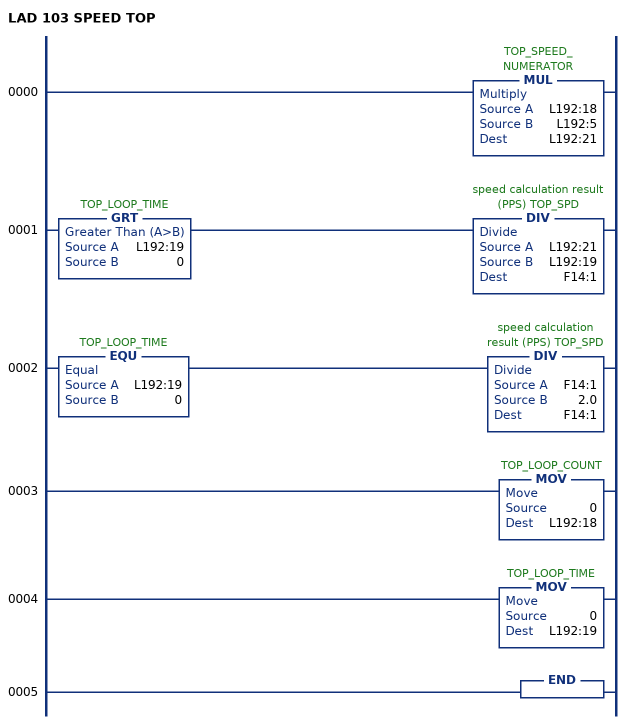
% Rung: 0 %
SOR MUL L192:18 L192:5 L192:21 EOR
%   L192:18  TOP_LOOP_COUNT %
%   L192:5  TKS_PER_SECOND %
%   L192:21  TOP_SPEED_NUMERATOR %
% Rung: 1 %
SOR GRT L192:19 0 DIV L192:21 L192:19 F14:1 EOR
%   L192:19  TOP_LOOP_TIME %
%   L192:21  TOP_SPEED_NUMERATOR %
%   F14:1  TOP_SPD  "speed calculation result (PPS)" %
% Rung: 2 %
SOR EQU L192:19 0 DIV F14:1 2.0 F14:1 EOR
%   L192:19  TOP_LOOP_TIME %
%   F14:1  TOP_SPD  "speed calculation result (PPS)" %
% Rung: 3 %
SOR MOV 0 L192:18 EOR
%   L192:18  TOP_LOOP_COUNT %
% Rung: 4 %
SOR MOV 0 L192:19 EOR
%   L192:19  TOP_LOOP_TIME %
% Rung: 5 %
SOR END EOR

LADDER 104 "P BOT"    % high speed %
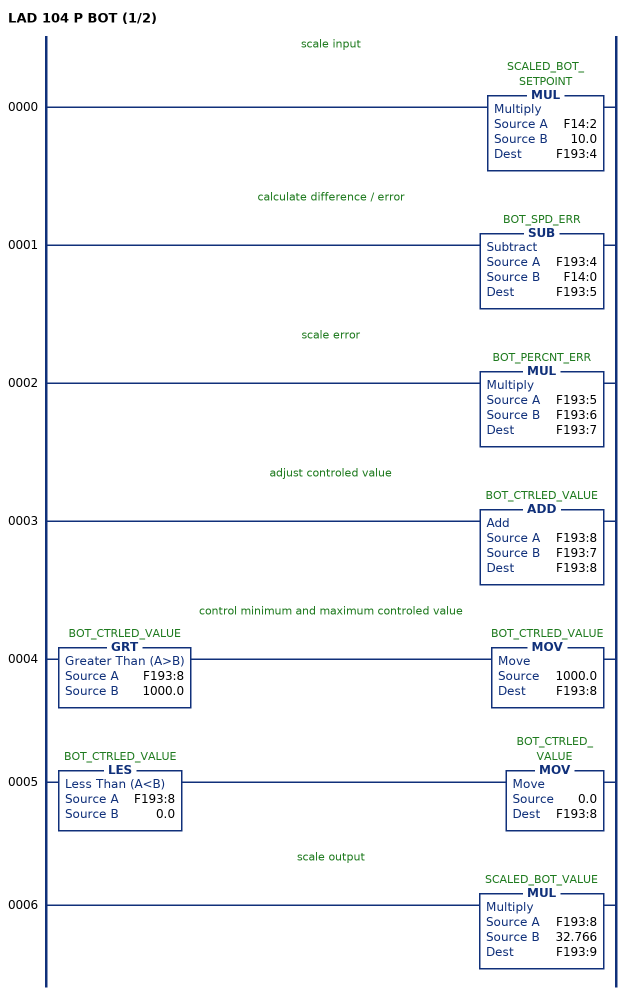
% Rung: 0 %
% scale input %
SOR MUL F14:2 10.0 F193:4 EOR
%   F14:2  BOT_SPD_SETPOINT %
%   F193:4  SCALED_BOT_SETPOINT %
% Rung: 1 %
% calculate difference / error %
SOR SUB F193:4 F14:0 F193:5 EOR
%   F193:4  SCALED_BOT_SETPOINT %
%   F14:0  BOT_SPD  "speed calculation result (PPS)" %
%   F193:5  BOT_SPD_ERR %
% Rung: 2 %
% scale error %
SOR MUL F193:5 F193:6 F193:7 EOR
%   F193:5  BOT_SPD_ERR %
%   F193:6  BOT_FDBK_RATIO %
%   F193:7  BOT_PERCNT_ERR %
% Rung: 3 %
% adjust controled value %
SOR ADD F193:8 F193:7 F193:8 EOR
%   F193:8  BOT_CTRLED_VALUE %
%   F193:7  BOT_PERCNT_ERR %
% Rung: 4 %
% control minimum and maximum controled value %
SOR GRT F193:8 1000.0 MOV 1000.0 F193:8 EOR
%   F193:8  BOT_CTRLED_VALUE %
% Rung: 5 %
SOR LES F193:8 0.0 MOV 0.0 F193:8 EOR
%   F193:8  BOT_CTRLED_VALUE %
% Rung: 6 %
% scale output %
SOR MUL F193:8 32.766 F193:9 EOR
%   F193:8  BOT_CTRLED_VALUE %
%   F193:9  SCALED_BOT_VALUE %

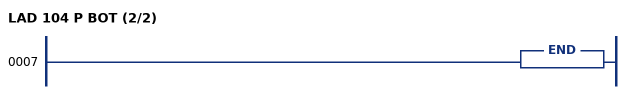
% Rung: 7 %
SOR END EOR

LADDER 105 "P TOP"    % high speed %
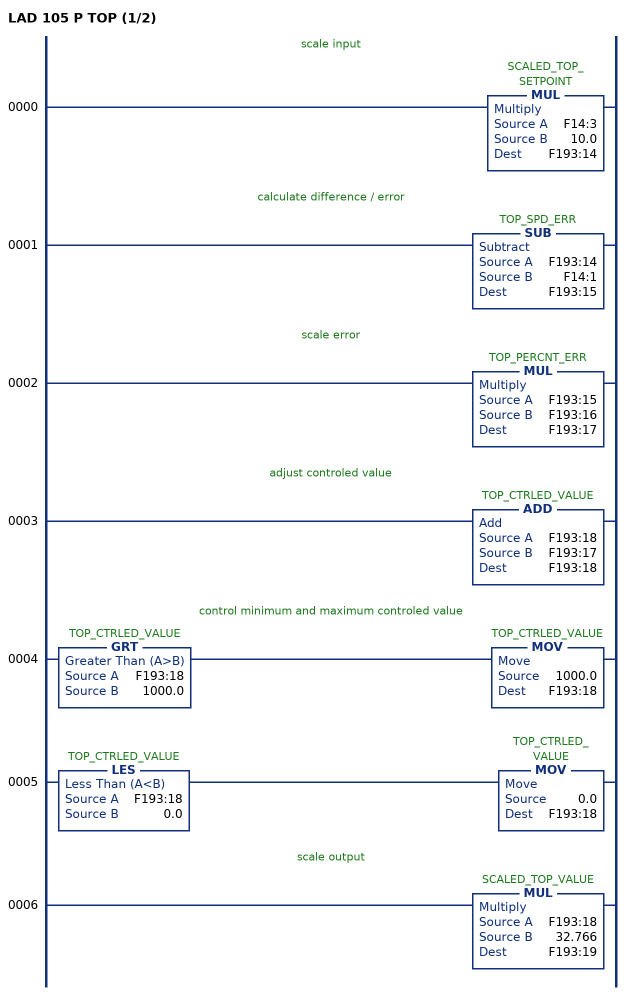
% Rung: 0 %
% scale input %
SOR MUL F14:3 10.0 F193:14 EOR
%   F14:3  TOP_SPD_SETPOINT %
%   F193:14  SCALED_TOP_SETPOINT %
% Rung: 1 %
% calculate difference / error %
SOR SUB F193:14 F14:1 F193:15 EOR
%   F193:14  SCALED_TOP_SETPOINT %
%   F14:1  TOP_SPD  "speed calculation result (PPS)" %
%   F193:15  TOP_SPD_ERR %
% Rung: 2 %
% scale error %
SOR MUL F193:15 F193:16 F193:17 EOR
%   F193:15  TOP_SPD_ERR %
%   F193:16  TOP_FDBK_RATIO %
%   F193:17  TOP_PERCNT_ERR %
% Rung: 3 %
% adjust controled value %
SOR ADD F193:18 F193:17 F193:18 EOR
%   F193:18  TOP_CTRLED_VALUE %
%   F193:17  TOP_PERCNT_ERR %
% Rung: 4 %
% control minimum and maximum controled value %
SOR GRT F193:18 1000.0 MOV 1000.0 F193:18 EOR
%   F193:18  TOP_CTRLED_VALUE %
% Rung: 5 %
SOR LES F193:18 0.0 MOV 0.0 F193:18 EOR
%   F193:18  TOP_CTRLED_VALUE %
% Rung: 6 %
% scale output %
SOR MUL F193:18 32.766 F193:19 EOR
%   F193:18  TOP_CTRLED_VALUE %
%   F193:19  SCALED_TOP_VALUE %

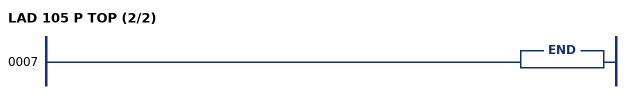
% Rung: 7 %
SOR END EOR

LADDER 110 "SHIFT BOT"
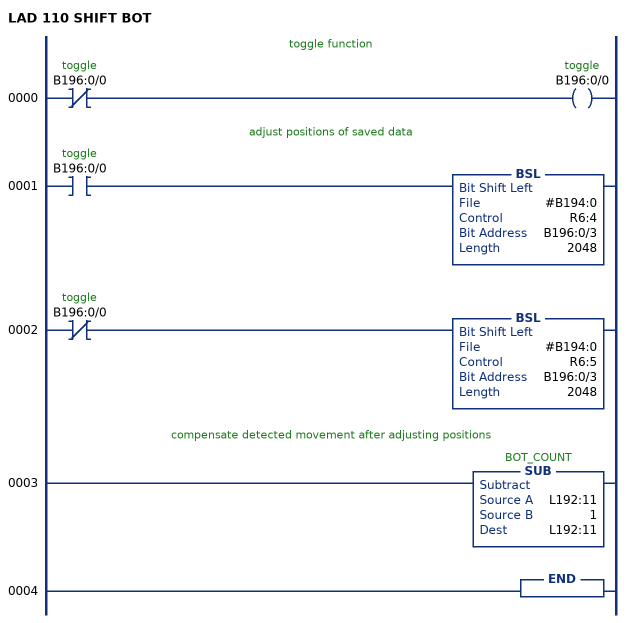
% Rung: 0 %
% toggle function %
SOR XIO B196:0/0 OTE B196:0/0 EOR
%   B196:0/0  "toggle" %
% Rung: 1 %
% adjust positions of saved data %
SOR XIC B196:0/0 BSL #B194:0 R6:4 B196:0/3 2048 EOR
%   B196:0/0  "toggle" %
%   B196:0/3  OFF %
% Rung: 2 %
SOR XIO B196:0/0 BSL #B194:0 R6:5 B196:0/3 2048 EOR
%   B196:0/0  "toggle" %
%   B196:0/3  OFF %
% Rung: 3 %
% compensate detected movement after adjusting positions %
SOR SUB L192:11 1 L192:11 EOR
%   L192:11  BOT_COUNT %
% Rung: 4 %
SOR END EOR

LADDER 111 "SHIFT TOP"
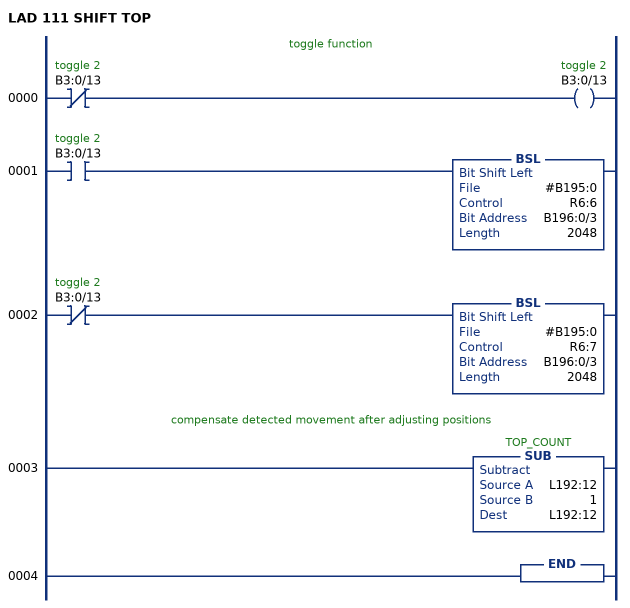
% Rung: 0 %
% toggle function %
SOR XIO B3:0/13 OTE B3:0/13 EOR
%   B3:0/13  "toggle 2" %
% Rung: 1 %
SOR XIC B3:0/13 BSL #B195:0 R6:6 B196:0/3 2048 EOR
%   B3:0/13  "toggle 2" %
%   B196:0/3  OFF %
% Rung: 2 %
SOR XIO B3:0/13 BSL #B195:0 R6:7 B196:0/3 2048 EOR
%   B3:0/13  "toggle 2" %
%   B196:0/3  OFF %
% Rung: 3 %
% compensate detected movement after adjusting positions %
SOR SUB L192:12 1 L192:12 EOR
%   L192:12  TOP_COUNT %
% Rung: 4 %
SOR END EOR

LADDER 122 "OPTICBOT"
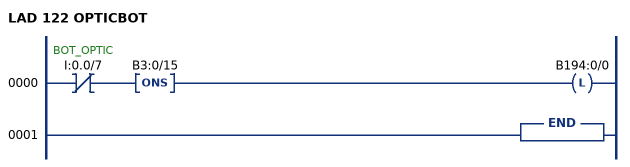
% Rung: 0 %
SOR XIO I:0.0/7 ONS B3:0/15 OTL B194:0/0 EOR
%   I:0.0/7  BOT_OPTIC %
% Rung: 1 %
SOR END EOR

LADDER 125 "INS 1TIME"
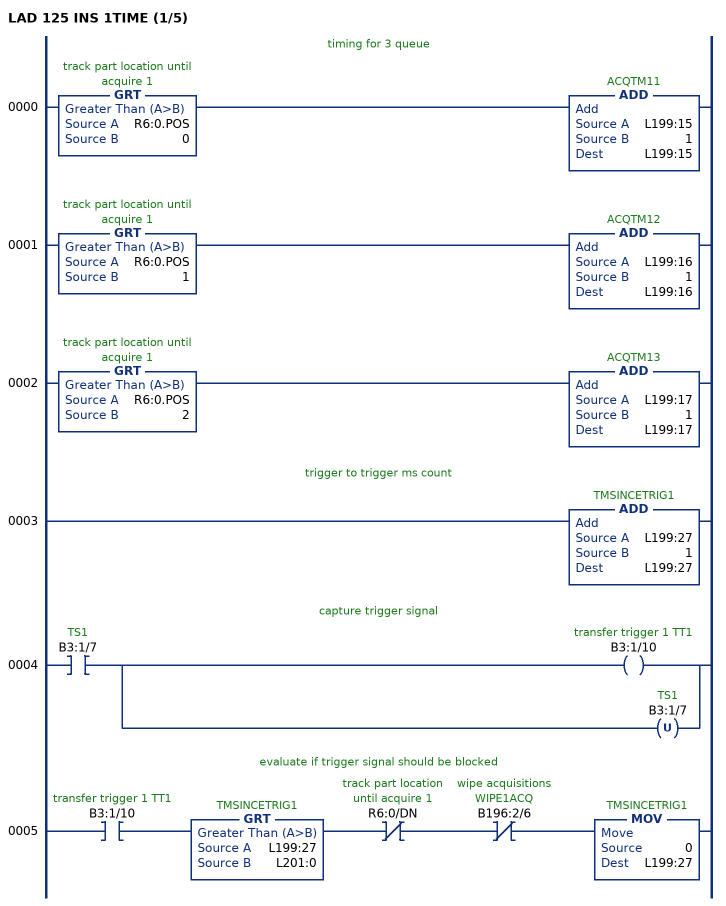
% Rung: 0 %
% timing for 3 queue %
SOR GRT R6:0.POS 0 ADD L199:15 1 L199:15 EOR
%   R6:0  "track part location until acquire 1" %
%   L199:15  ACQTM11 %
% Rung: 1 %
SOR GRT R6:0.POS 1 ADD L199:16 1 L199:16 EOR
%   R6:0  "track part location until acquire 1" %
%   L199:16  ACQTM12 %
% Rung: 2 %
SOR GRT R6:0.POS 2 ADD L199:17 1 L199:17 EOR
%   R6:0  "track part location until acquire 1" %
%   L199:17  ACQTM13 %
% Rung: 3 %
% trigger to trigger ms count %
SOR ADD L199:27 1 L199:27 EOR
%   L199:27  TMSINCETRIG1 %
% Rung: 4 %
% capture trigger signal %
SOR XIC B3:1/7 BST OTE B3:1/10 NXB OTU B3:1/7 BND EOR
%   B3:1/7  TS1 %
%   B3:1/10  TT1  "transfer trigger 1" %
% Rung: 5 %
% evaluate if trigger signal should be blocked %
SOR XIC B3:1/10 GRT L199:27 L201:0 XIO R6:0/DN XIO B196:2/6 MOV 0 L199:27 EOR
%   B3:1/10  TT1  "transfer trigger 1" %
%   L199:27  TMSINCETRIG1 %
%   L201:0  CAM_1_MIN_CY %
%   R6:0  "track part location until acquire 1" %
%   B196:2/6  WIPE1ACQ  "wipe acquisitions" %

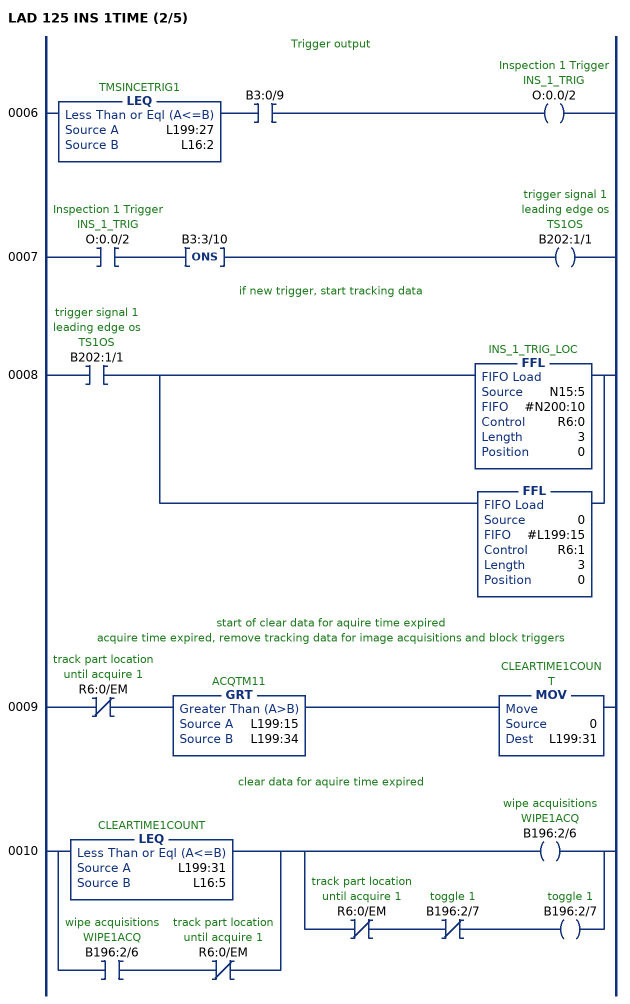
% Rung: 6 %
% Trigger output %
SOR LEQ L199:27 L16:2 XIC B3:0/9 OTE O:0.0/2 EOR
%   L199:27  TMSINCETRIG1 %
%   L16:2  CAM_1_TRIG_TIME %
%   O:0.0/2  INS_1_TRIG  "Inspection 1 Trigger" %
% Rung: 7 %
SOR XIC O:0.0/2 ONS B3:3/10 OTE B202:1/1 EOR
%   O:0.0/2  INS_1_TRIG  "Inspection 1 Trigger" %
%   B202:1/1  TS1OS  "trigger signal 1 leading edge os" %
% Rung: 8 %
% if new trigger, start tracking data %
SOR XIC B202:1/1 BST FFL N15:5 #N200:10 R6:0 3 0 NXB FFL 0 #L199:15 R6:1 3 0 BND EOR
%   B202:1/1  TS1OS  "trigger signal 1 leading edge os" %
%   N15:5  INS_1_TRIG_LOC %
%   N200:10  ACQPOS11 %
%   R6:0  "track part location until acquire 1" %
%   L199:15  ACQTM11 %
%   R6:1  "track acquire time 1" %
% Rung: 9 %
% start of clear data for aquire time expired
% acquire time expired, remove tracking data for image acquisitions and block triggers %
SOR XIO R6:0/EM GRT L199:15 L199:34 MOV 0 L199:31 EOR
%   R6:0  "track part location until acquire 1" %
%   L199:15  ACQTM11 %
%   L199:34  MAXACQTM1 %
%   L199:31  CLEARTIME1COUNT %
% Rung: 10 %
% clear data for aquire time expired %
SOR BST LEQ L199:31 L16:5 NXB XIC B196:2/6 XIO R6:0/EM BND BST OTE B196:2/6 NXB XIO R6:0/EM XIO B196:2/7 OTE B196:2/7 BND EOR
%   L199:31  CLEARTIME1COUNT %
%   L16:5  CLEARTIME1  "time to clear tracking data" %
%   B196:2/6  WIPE1ACQ  "wipe acquisitions" %
%   R6:0  "track part location until acquire 1" %
%   B196:2/7  "toggle 1" %

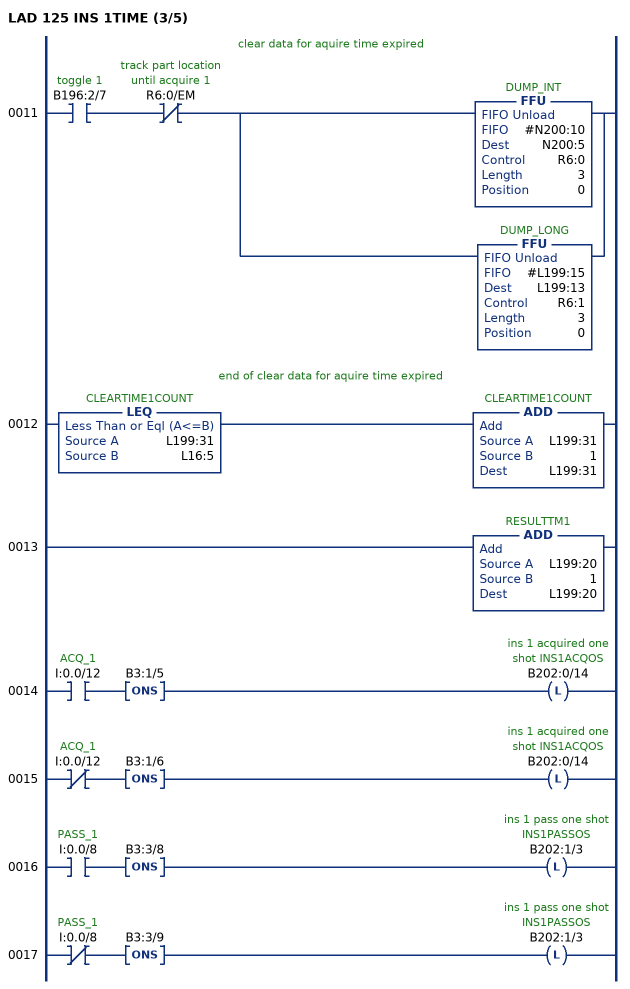
% Rung: 11 %
% clear data for aquire time expired %
SOR XIC B196:2/7 XIO R6:0/EM BST FFU #N200:10 N200:5 R6:0 3 0 NXB FFU #L199:15 L199:13 R6:1 3 0 BND EOR
%   B196:2/7  "toggle 1" %
%   R6:0  "track part location until acquire 1" %
%   N200:10  ACQPOS11 %
%   N200:5  DUMP_INT %
%   L199:15  ACQTM11 %
%   L199:13  DUMP_LONG %
%   R6:1  "track acquire time 1" %
% Rung: 12 %
% end of clear data for aquire time expired %
SOR LEQ L199:31 L16:5 ADD L199:31 1 L199:31 EOR
%   L199:31  CLEARTIME1COUNT %
%   L16:5  CLEARTIME1  "time to clear tracking data" %
% Rung: 13 %
SOR ADD L199:20 1 L199:20 EOR
%   L199:20  RESULTTM1 %
% Rung: 14 %
SOR XIC I:0.0/12 ONS B3:1/5 OTL B202:0/14 EOR
%   I:0.0/12  ACQ_1 %
%   B202:0/14  INS1ACQOS  "ins 1 acquired one shot" %
% Rung: 15 %
SOR XIO I:0.0/12 ONS B3:1/6 OTL B202:0/14 EOR
%   I:0.0/12  ACQ_1 %
%   B202:0/14  INS1ACQOS  "ins 1 acquired one shot" %
% Rung: 16 %
SOR XIC I:0.0/8 ONS B3:3/8 OTL B202:1/3 EOR
%   I:0.0/8  PASS_1 %
%   B202:1/3  INS1PASSOS  "ins 1 pass one shot" %
% Rung: 17 %
SOR XIO I:0.0/8 ONS B3:3/9 OTL B202:1/3 EOR
%   I:0.0/8  PASS_1 %
%   B202:1/3  INS1PASSOS  "ins 1 pass one shot" %

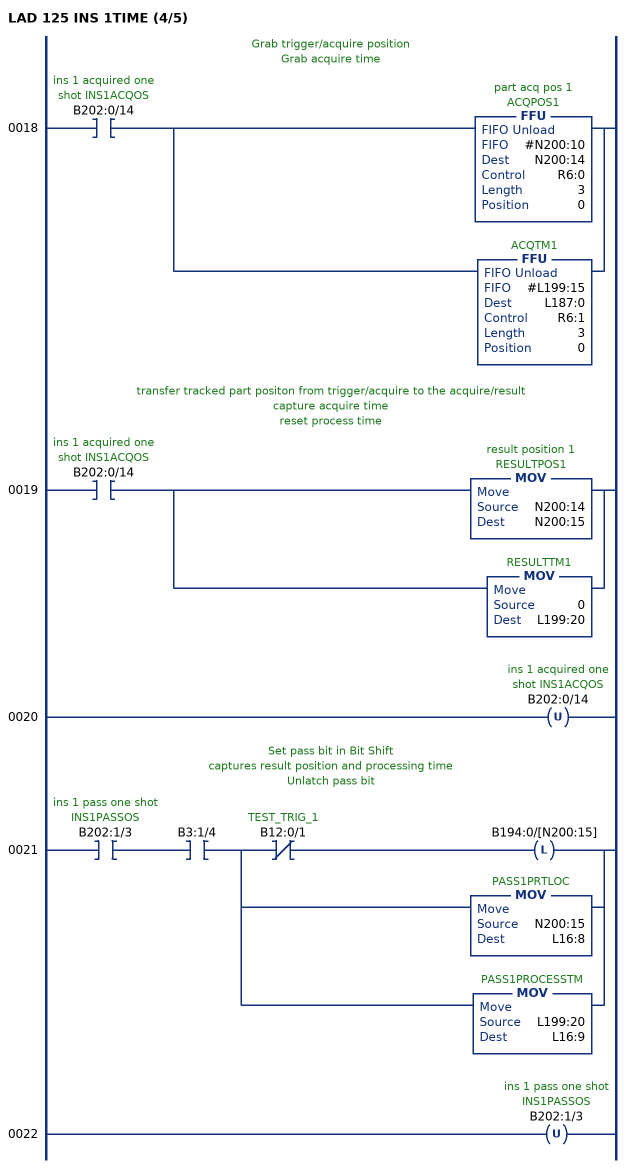
% Rung: 18 %
% Grab trigger/acquire position
% Grab acquire time %
SOR XIC B202:0/14 BST FFU #N200:10 N200:14 R6:0 3 0 NXB FFU #L199:15 L187:0 R6:1 3 0 BND EOR
%   B202:0/14  INS1ACQOS  "ins 1 acquired one shot" %
%   N200:10  ACQPOS11 %
%   N200:14  ACQPOS1  "part acq pos 1" %
%   R6:0  "track part location until acquire 1" %
%   L199:15  ACQTM11 %
%   L187:0  ACQTM1 %
%   R6:1  "track acquire time 1" %
% Rung: 19 %
% transfer tracked part positon from trigger/acquire to the acquire/result
% capture acquire time
% reset process time %
SOR XIC B202:0/14 BST MOV N200:14 N200:15 NXB MOV 0 L199:20 BND EOR
%   B202:0/14  INS1ACQOS  "ins 1 acquired one shot" %
%   N200:14  ACQPOS1  "part acq pos 1" %
%   N200:15  RESULTPOS1  "result position 1" %
%   L199:20  RESULTTM1 %
% Rung: 20 %
SOR OTU B202:0/14 EOR
%   B202:0/14  INS1ACQOS  "ins 1 acquired one shot" %
% Rung: 21 %
% Set pass bit in Bit Shift
% captures result position and processing time
% Unlatch pass bit %
SOR XIC B202:1/3 XIC B3:1/4 BST XIO B12:0/1 OTL B194:0/[N200:15] NXB MOV N200:15 L16:8 NXB MOV L199:20 L16:9 BND EOR
%   B202:1/3  INS1PASSOS  "ins 1 pass one shot" %
%   B12:0/1  TEST_TRIG_1 %
%   N200:15  RESULTPOS1  "result position 1" %
%   L16:8  PASS1PRTLOC %
%   L199:20  RESULTTM1 %
%   L16:9  PASS1PROCESSTM %
% Rung: 22 %
SOR OTU B202:1/3 EOR
%   B202:1/3  INS1PASSOS  "ins 1 pass one shot" %

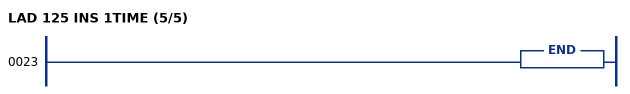
% Rung: 23 %
SOR END EOR

LADDER 126 "INS 1 MOVE"
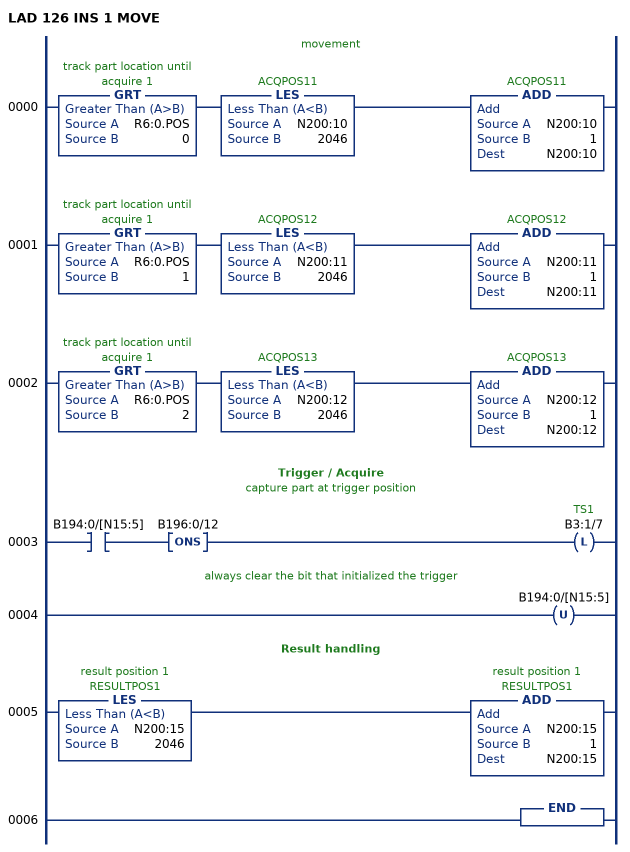
% Rung: 0 %
% movement %
SOR GRT R6:0.POS 0 LES N200:10 2046 ADD N200:10 1 N200:10 EOR
%   R6:0  "track part location until acquire 1" %
%   N200:10  ACQPOS11 %
% Rung: 1 %
SOR GRT R6:0.POS 1 LES N200:11 2046 ADD N200:11 1 N200:11 EOR
%   R6:0  "track part location until acquire 1" %
%   N200:11  ACQPOS12 %
% Rung: 2 %
SOR GRT R6:0.POS 2 LES N200:12 2046 ADD N200:12 1 N200:12 EOR
%   R6:0  "track part location until acquire 1" %
%   N200:12  ACQPOS13 %
% Rung: 3 %
% TITLE: Trigger / Acquire %
% capture part at trigger position %
SOR XIC B194:0/[N15:5] ONS B196:0/12 OTL B3:1/7 EOR
%   N15:5  INS_1_TRIG_LOC %
%   B3:1/7  TS1 %
% Rung: 4 %
% always clear the bit that initialized the trigger %
SOR OTU B194:0/[N15:5] EOR
%   N15:5  INS_1_TRIG_LOC %
% Rung: 5 %
% TITLE: Result handling %
SOR LES N200:15 2046 ADD N200:15 1 N200:15 EOR
%   N200:15  RESULTPOS1  "result position 1" %
% Rung: 6 %
SOR END EOR

LADDER 131 "XFER"
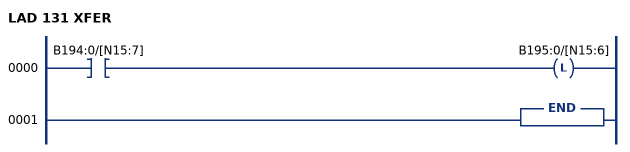
% Rung: 0 %
SOR XIC B194:0/[N15:7] OTL B195:0/[N15:6] EOR
%   N15:7  XFER_OUT_LOC %
%   N15:6  XFER_IN_LOC %
% Rung: 1 %
SOR END EOR

LADDER 141 "OPTICTOP"
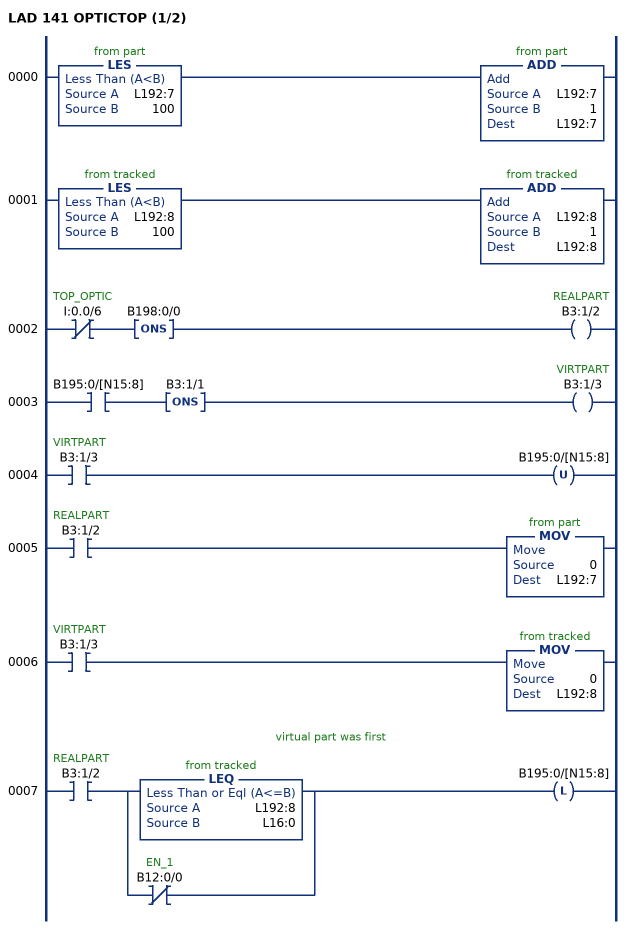
% Rung: 0 %
SOR LES L192:7 100 ADD L192:7 1 L192:7 EOR
%   L192:7  "from part" %
% Rung: 1 %
SOR LES L192:8 100 ADD L192:8 1 L192:8 EOR
%   L192:8  "from tracked" %
% Rung: 2 %
SOR XIO I:0.0/6 ONS B198:0/0 OTE B3:1/2 EOR
%   I:0.0/6  TOP_OPTIC %
%   B3:1/2  REALPART %
% Rung: 3 %
SOR XIC B195:0/[N15:8] ONS B3:1/1 OTE B3:1/3 EOR
%   N15:8  TOP_OPTIC_LOC %
%   B3:1/3  VIRTPART %
% Rung: 4 %
SOR XIC B3:1/3 OTU B195:0/[N15:8] EOR
%   B3:1/3  VIRTPART %
%   N15:8  TOP_OPTIC_LOC %
% Rung: 5 %
SOR XIC B3:1/2 MOV 0 L192:7 EOR
%   B3:1/2  REALPART %
%   L192:7  "from part" %
% Rung: 6 %
SOR XIC B3:1/3 MOV 0 L192:8 EOR
%   B3:1/3  VIRTPART %
%   L192:8  "from tracked" %
% Rung: 7 %
% virtual part was first %
SOR XIC B3:1/2 BST LEQ L192:8 L16:0 NXB XIO B12:0/0 BND OTL B195:0/[N15:8] EOR
%   B3:1/2  REALPART %
%   L192:8  "from tracked" %
%   B12:0/0  EN_1 %
%   N15:8  TOP_OPTIC_LOC %

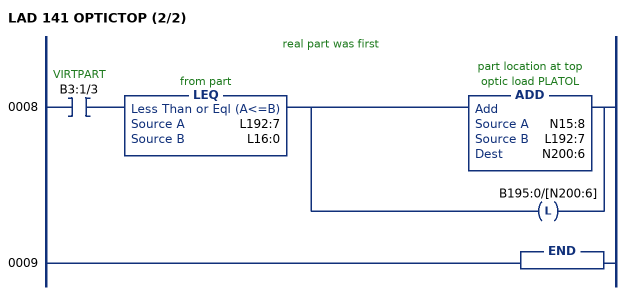
% Rung: 8 %
% real part was first %
SOR XIC B3:1/3 LEQ L192:7 L16:0 BST ADD N15:8 L192:7 N200:6 NXB OTL B195:0/[N200:6] BND EOR
%   B3:1/3  VIRTPART %
%   L192:7  "from part" %
%   N15:8  TOP_OPTIC_LOC %
%   N200:6  PLATOL  "part location at top optic load" %
% Rung: 9 %
SOR END EOR

LADDER 150 "INS 5 TIME"
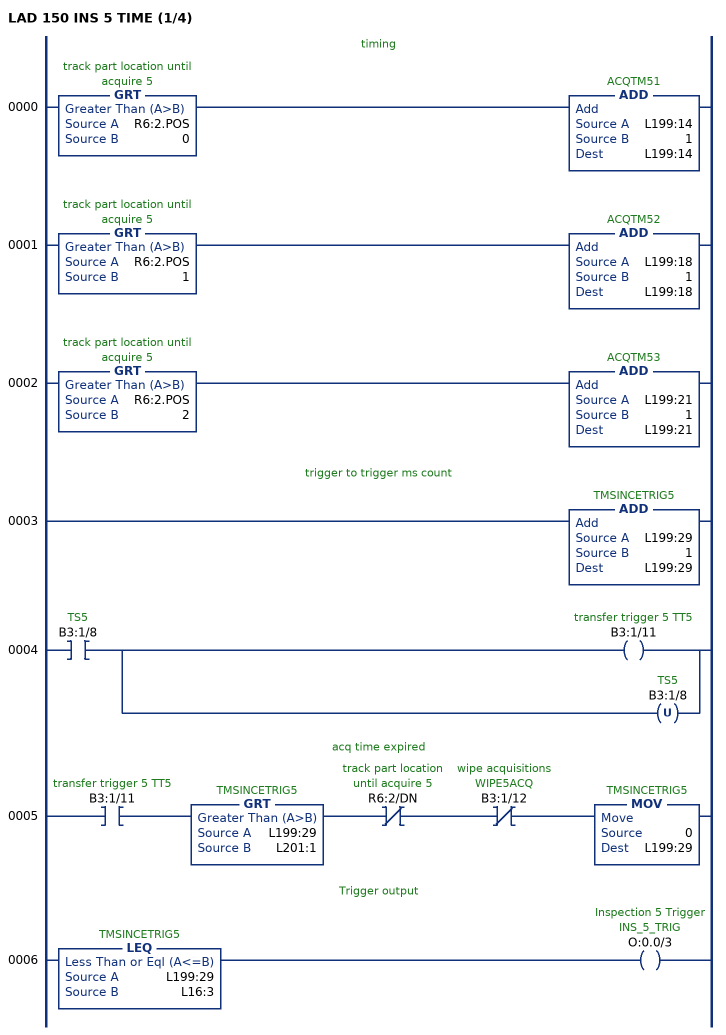
% Rung: 0 %
% timing %
SOR GRT R6:2.POS 0 ADD L199:14 1 L199:14 EOR
%   R6:2  "track part location until acquire 5" %
%   L199:14  ACQTM51 %
% Rung: 1 %
SOR GRT R6:2.POS 1 ADD L199:18 1 L199:18 EOR
%   R6:2  "track part location until acquire 5" %
%   L199:18  ACQTM52 %
% Rung: 2 %
SOR GRT R6:2.POS 2 ADD L199:21 1 L199:21 EOR
%   R6:2  "track part location until acquire 5" %
%   L199:21  ACQTM53 %
% Rung: 3 %
% trigger to trigger ms count %
SOR ADD L199:29 1 L199:29 EOR
%   L199:29  TMSINCETRIG5 %
% Rung: 4 %
SOR XIC B3:1/8 BST OTE B3:1/11 NXB OTU B3:1/8 BND EOR
%   B3:1/8  TS5 %
%   B3:1/11  TT5  "transfer trigger 5" %
% Rung: 5 %
% acq time expired %
SOR XIC B3:1/11 GRT L199:29 L201:1 XIO R6:2/DN XIO B3:1/12 MOV 0 L199:29 EOR
%   B3:1/11  TT5  "transfer trigger 5" %
%   L199:29  TMSINCETRIG5 %
%   L201:1  CAM_5_MIN_CY %
%   R6:2  "track part location until acquire 5" %
%   B3:1/12  WIPE5ACQ  "wipe acquisitions" %
% Rung: 6 %
% Trigger output %
SOR LEQ L199:29 L16:3 OTE O:0.0/3 EOR
%   L199:29  TMSINCETRIG5 %
%   L16:3  CAM_5_TRIG_TIME %
%   O:0.0/3  INS_5_TRIG  "Inspection 5 Trigger" %

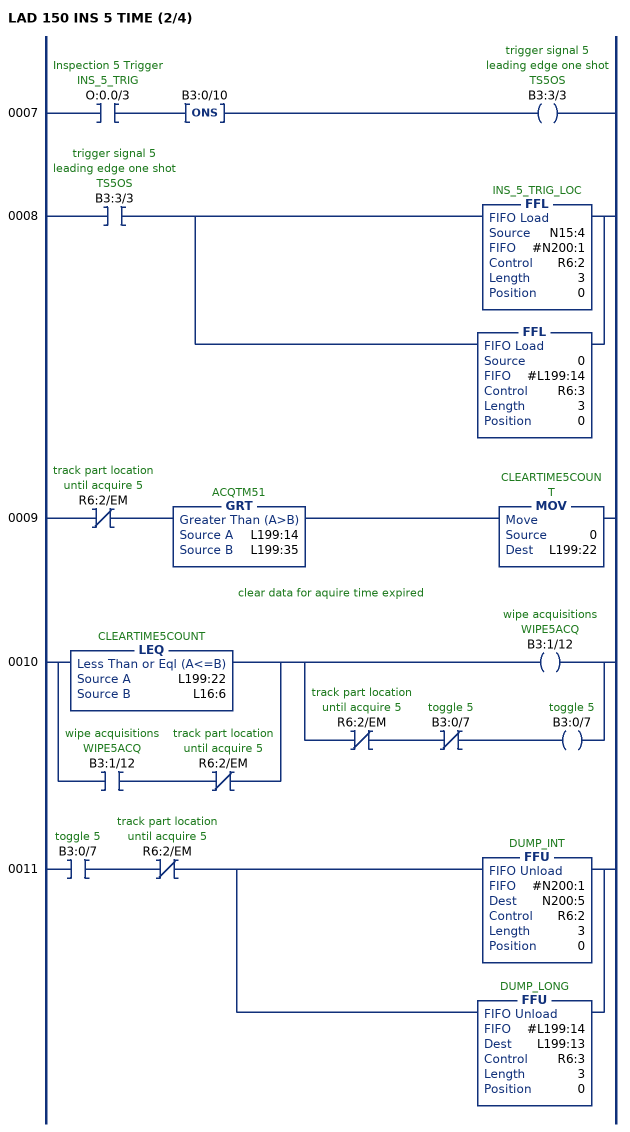
% Rung: 7 %
SOR XIC O:0.0/3 ONS B3:0/10 OTE B3:3/3 EOR
%   O:0.0/3  INS_5_TRIG  "Inspection 5 Trigger" %
%   B3:3/3  TS5OS  "trigger signal 5 leading edge one shot" %
% Rung: 8 %
SOR XIC B3:3/3 BST FFL N15:4 #N200:1 R6:2 3 0 NXB FFL 0 #L199:14 R6:3 3 0 BND EOR
%   B3:3/3  TS5OS  "trigger signal 5 leading edge one shot" %
%   N15:4  INS_5_TRIG_LOC %
%   N200:1  ACQPOS51 %
%   R6:2  "track part location until acquire 5" %
%   L199:14  ACQTM51 %
%   R6:3  "track acquire time 5" %
% Rung: 9 %
SOR XIO R6:2/EM GRT L199:14 L199:35 MOV 0 L199:22 EOR
%   R6:2  "track part location until acquire 5" %
%   L199:14  ACQTM51 %
%   L199:35  MAXACQTM5 %
%   L199:22  CLEARTIME5COUNT %
% Rung: 10 %
% clear data for aquire time expired %
SOR BST LEQ L199:22 L16:6 NXB XIC B3:1/12 XIO R6:2/EM BND BST OTE B3:1/12 NXB XIO R6:2/EM XIO B3:0/7 OTE B3:0/7 BND EOR
%   L199:22  CLEARTIME5COUNT %
%   L16:6  CLEARTIME5 %
%   B3:1/12  WIPE5ACQ  "wipe acquisitions" %
%   R6:2  "track part location until acquire 5" %
%   B3:0/7  "toggle 5" %
% Rung: 11 %
SOR XIC B3:0/7 XIO R6:2/EM BST FFU #N200:1 N200:5 R6:2 3 0 NXB FFU #L199:14 L199:13 R6:3 3 0 BND EOR
%   B3:0/7  "toggle 5" %
%   R6:2  "track part location until acquire 5" %
%   N200:1  ACQPOS51 %
%   N200:5  DUMP_INT %
%   L199:14  ACQTM51 %
%   L199:13  DUMP_LONG %
%   R6:3  "track acquire time 5" %

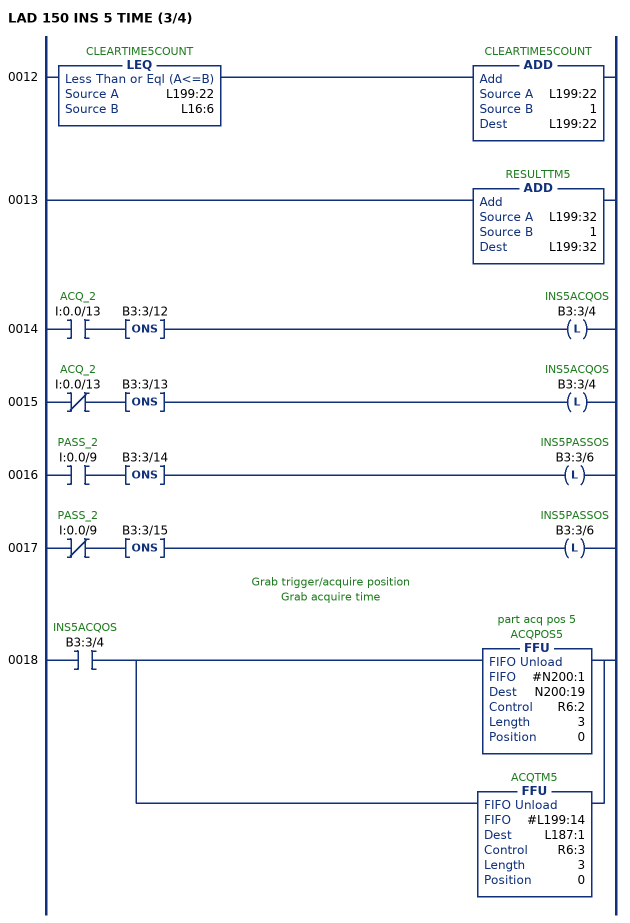
% Rung: 12 %
SOR LEQ L199:22 L16:6 ADD L199:22 1 L199:22 EOR
%   L199:22  CLEARTIME5COUNT %
%   L16:6  CLEARTIME5 %
% Rung: 13 %
SOR ADD L199:32 1 L199:32 EOR
%   L199:32  RESULTTM5 %
% Rung: 14 %
SOR XIC I:0.0/13 ONS B3:3/12 OTL B3:3/4 EOR
%   I:0.0/13  ACQ_2 %
%   B3:3/4  INS5ACQOS %
% Rung: 15 %
SOR XIO I:0.0/13 ONS B3:3/13 OTL B3:3/4 EOR
%   I:0.0/13  ACQ_2 %
%   B3:3/4  INS5ACQOS %
% Rung: 16 %
SOR XIC I:0.0/9 ONS B3:3/14 OTL B3:3/6 EOR
%   I:0.0/9  PASS_2 %
%   B3:3/6  INS5PASSOS %
% Rung: 17 %
SOR XIO I:0.0/9 ONS B3:3/15 OTL B3:3/6 EOR
%   I:0.0/9  PASS_2 %
%   B3:3/6  INS5PASSOS %
% Rung: 18 %
% Grab trigger/acquire position
% Grab acquire time %
SOR XIC B3:3/4 BST FFU #N200:1 N200:19 R6:2 3 0 NXB FFU #L199:14 L187:1 R6:3 3 0 BND EOR
%   B3:3/4  INS5ACQOS %
%   N200:1  ACQPOS51 %
%   N200:19  ACQPOS5  "part acq pos 5" %
%   R6:2  "track part location until acquire 5" %
%   L199:14  ACQTM51 %
%   L187:1  ACQTM5 %
%   R6:3  "track acquire time 5" %

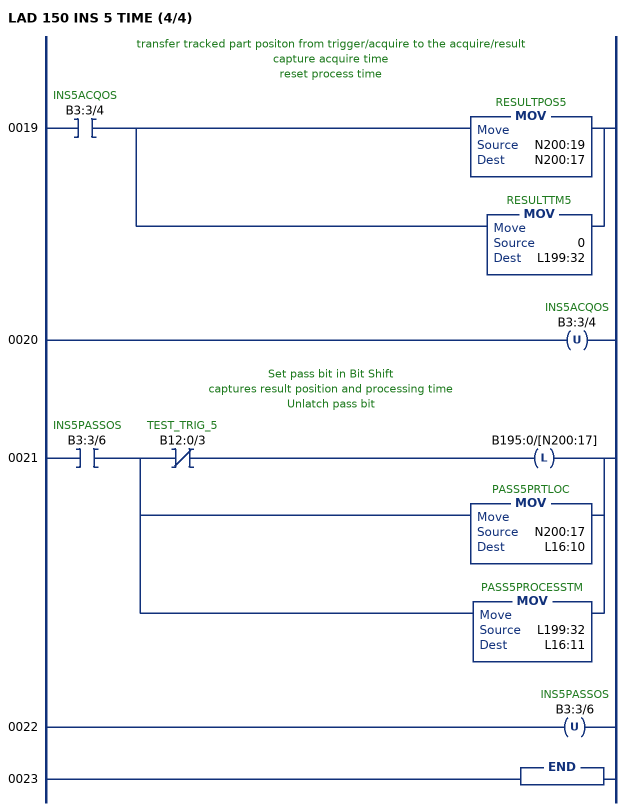
% Rung: 19 %
% transfer tracked part positon from trigger/acquire to the acquire/result
% capture acquire time
% reset process time %
SOR XIC B3:3/4 BST MOV N200:19 N200:17 NXB MOV 0 L199:32 BND EOR
%   B3:3/4  INS5ACQOS %
%   N200:19  ACQPOS5  "part acq pos 5" %
%   N200:17  RESULTPOS5 %
%   L199:32  RESULTTM5 %
% Rung: 20 %
SOR OTU B3:3/4 EOR
%   B3:3/4  INS5ACQOS %
% Rung: 21 %
% Set pass bit in Bit Shift
% captures result position and processing time
% Unlatch pass bit %
SOR XIC B3:3/6 BST XIO B12:0/3 OTL B195:0/[N200:17] NXB MOV N200:17 L16:10 NXB MOV L199:32 L16:11 BND EOR
%   B3:3/6  INS5PASSOS %
%   B12:0/3  TEST_TRIG_5 %
%   N200:17  RESULTPOS5 %
%   L16:10  PASS5PRTLOC %
%   L199:32  RESULTTM5 %
%   L16:11  PASS5PROCESSTM %
% Rung: 22 %
SOR OTU B3:3/6 EOR
%   B3:3/6  INS5PASSOS %
% Rung: 23 %
SOR END EOR

LADDER 151 "INS 5 MOVE"
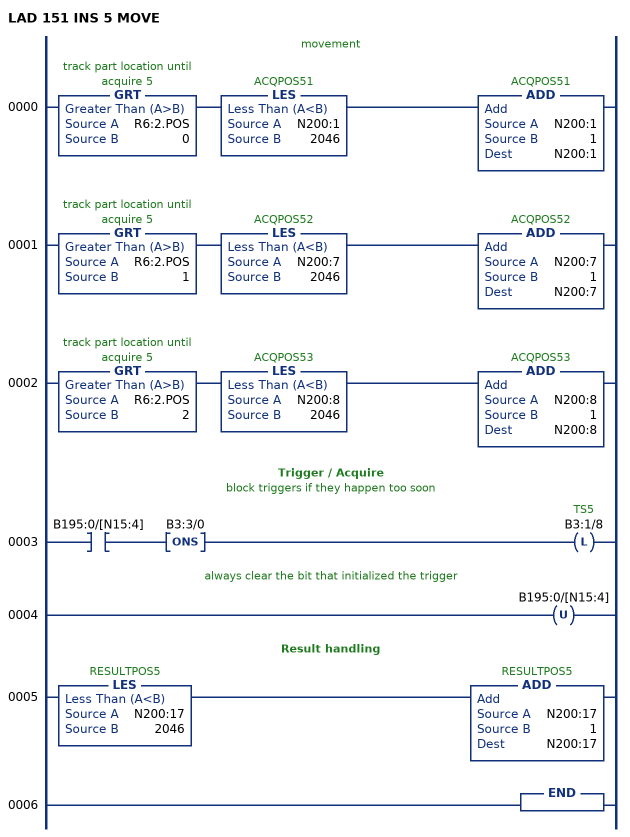
% Rung: 0 %
% movement %
SOR GRT R6:2.POS 0 LES N200:1 2046 ADD N200:1 1 N200:1 EOR
%   R6:2  "track part location until acquire 5" %
%   N200:1  ACQPOS51 %
% Rung: 1 %
SOR GRT R6:2.POS 1 LES N200:7 2046 ADD N200:7 1 N200:7 EOR
%   R6:2  "track part location until acquire 5" %
%   N200:7  ACQPOS52 %
% Rung: 2 %
SOR GRT R6:2.POS 2 LES N200:8 2046 ADD N200:8 1 N200:8 EOR
%   R6:2  "track part location until acquire 5" %
%   N200:8  ACQPOS53 %
% Rung: 3 %
% TITLE: Trigger / Acquire %
% block triggers if they happen too soon %
SOR XIC B195:0/[N15:4] ONS B3:3/0 OTL B3:1/8 EOR
%   N15:4  INS_5_TRIG_LOC %
%   B3:1/8  TS5 %
% Rung: 4 %
% always clear the bit that initialized the trigger %
SOR OTU B195:0/[N15:4] EOR
%   N15:4  INS_5_TRIG_LOC %
% Rung: 5 %
% TITLE: Result handling %
SOR LES N200:17 2046 ADD N200:17 1 N200:17 EOR
%   N200:17  RESULTPOS5 %
% Rung: 6 %
SOR END EOR

LADDER 160 "INS 6 TIME"
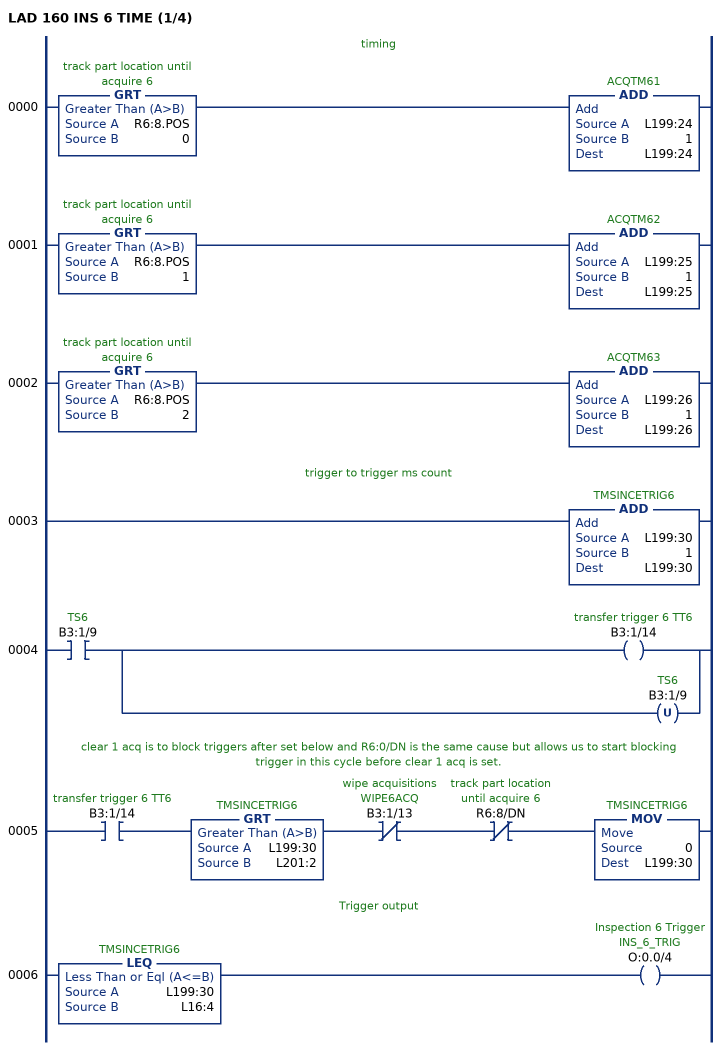
% Rung: 0 %
% timing %
SOR GRT R6:8.POS 0 ADD L199:24 1 L199:24 EOR
%   R6:8  "track part location until acquire 6" %
%   L199:24  ACQTM61 %
% Rung: 1 %
SOR GRT R6:8.POS 1 ADD L199:25 1 L199:25 EOR
%   R6:8  "track part location until acquire 6" %
%   L199:25  ACQTM62 %
% Rung: 2 %
SOR GRT R6:8.POS 2 ADD L199:26 1 L199:26 EOR
%   R6:8  "track part location until acquire 6" %
%   L199:26  ACQTM63 %
% Rung: 3 %
% trigger to trigger ms count %
SOR ADD L199:30 1 L199:30 EOR
%   L199:30  TMSINCETRIG6 %
% Rung: 4 %
SOR XIC B3:1/9 BST OTE B3:1/14 NXB OTU B3:1/9 BND EOR
%   B3:1/9  TS6 %
%   B3:1/14  TT6  "transfer trigger 6" %
% Rung: 5 %
% clear 1 acq is to block triggers after set below and R6:0/DN is the same cause but allows us to start blocking trigger in this cycle before clear 1 acq is set. %
SOR XIC B3:1/14 GRT L199:30 L201:2 XIO B3:1/13 XIO R6:8/DN MOV 0 L199:30 EOR
%   B3:1/14  TT6  "transfer trigger 6" %
%   L199:30  TMSINCETRIG6 %
%   L201:2  CAM_6_MIN_CY %
%   B3:1/13  WIPE6ACQ  "wipe acquisitions" %
%   R6:8  "track part location until acquire 6" %
% Rung: 6 %
% Trigger output %
SOR LEQ L199:30 L16:4 OTE O:0.0/4 EOR
%   L199:30  TMSINCETRIG6 %
%   L16:4  CAM_6_TRIG_TIME %
%   O:0.0/4  INS_6_TRIG  "Inspection 6 Trigger" %

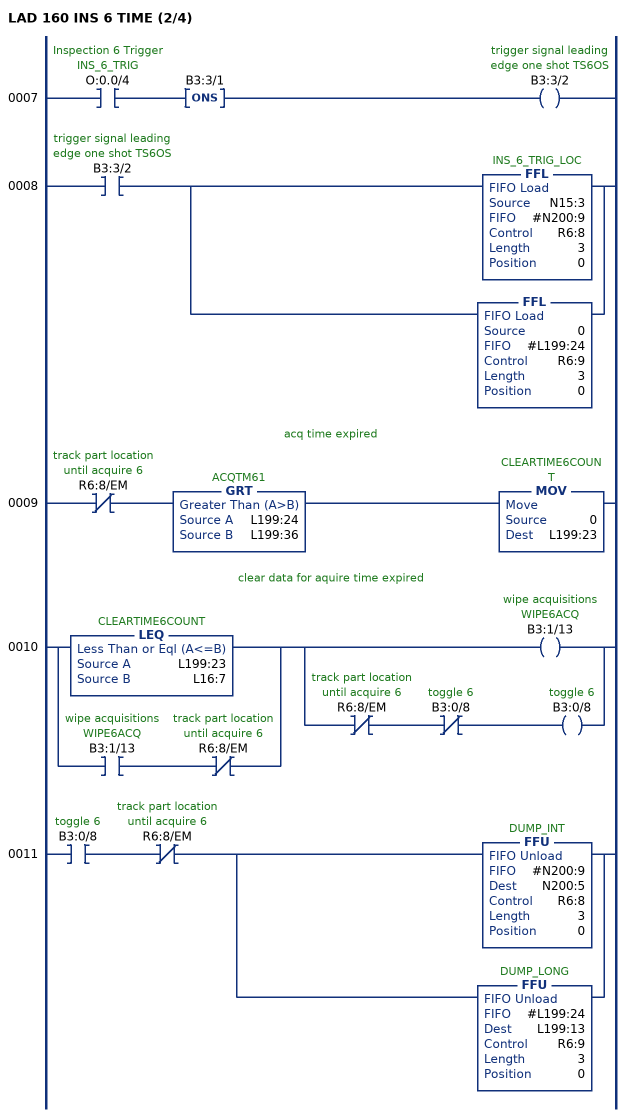
% Rung: 7 %
SOR XIC O:0.0/4 ONS B3:3/1 OTE B3:3/2 EOR
%   O:0.0/4  INS_6_TRIG  "Inspection 6 Trigger" %
%   B3:3/2  TS6OS  "trigger signal leading edge one shot" %
% Rung: 8 %
SOR XIC B3:3/2 BST FFL N15:3 #N200:9 R6:8 3 0 NXB FFL 0 #L199:24 R6:9 3 0 BND EOR
%   B3:3/2  TS6OS  "trigger signal leading edge one shot" %
%   N15:3  INS_6_TRIG_LOC %
%   N200:9  ACQPOS61 %
%   R6:8  "track part location until acquire 6" %
%   L199:24  ACQTM61 %
%   R6:9  "track acquire time 6" %
% Rung: 9 %
% acq time expired %
SOR XIO R6:8/EM GRT L199:24 L199:36 MOV 0 L199:23 EOR
%   R6:8  "track part location until acquire 6" %
%   L199:24  ACQTM61 %
%   L199:36  MAXACQTM6 %
%   L199:23  CLEARTIME6COUNT %
% Rung: 10 %
% clear data for aquire time expired %
SOR BST LEQ L199:23 L16:7 NXB XIC B3:1/13 XIO R6:8/EM BND BST OTE B3:1/13 NXB XIO R6:8/EM XIO B3:0/8 OTE B3:0/8 BND EOR
%   L199:23  CLEARTIME6COUNT %
%   L16:7  CLEARTIME6 %
%   B3:1/13  WIPE6ACQ  "wipe acquisitions" %
%   R6:8  "track part location until acquire 6" %
%   B3:0/8  "toggle 6" %
% Rung: 11 %
SOR XIC B3:0/8 XIO R6:8/EM BST FFU #N200:9 N200:5 R6:8 3 0 NXB FFU #L199:24 L199:13 R6:9 3 0 BND EOR
%   B3:0/8  "toggle 6" %
%   R6:8  "track part location until acquire 6" %
%   N200:9  ACQPOS61 %
%   N200:5  DUMP_INT %
%   L199:24  ACQTM61 %
%   L199:13  DUMP_LONG %
%   R6:9  "track acquire time 6" %

